{attribute 'qualified_only'}
TYPE E_CoatingStates :
(
    Unknown := 0,
    L0B4C := 1,
    L0Ni := 2,
    L0_L1B4C := 3,
    L0_L1Ni := 4
) UINT;
END_TYPE

(* stored: Version 1.1.0.1, ProductVersion 3.1.4022.18
   DUT E_CoatingStates: Id {118e1a24-82d2-4598-99ea-540bbe0bbd1a} *)
